Fanuc KAREL source: NC0056.KL

-- PROVISIONAL review KL for V940-1; original PC SHA256 2b6319c3cb2ebb61502ed711de4ec4e3f4f6b1a3b38024a92c039d9d4e8bd108
-- Incomplete behavior may be omitted. Consult companion uncertainty JSON. Do not deploy.
PROGRAM NC0056
%NOLOCKGROUP
-- UNRESOLVED_LOCAL_POOL 1 cells at code offset 3; source declarations unknown
-- DIRECT_LOCAL_WORD_ACCESS alone does not prove INTEGER, REAL, or BOOLEAN
BEGIN
  -- V9_CONDITION_STACK_HINT 4 bounded expression windows; static native code-base-relative target link; source arms held
  -- UNRESOLVED_PC offsets 0-8; opcodes 2B,2C,7B
  -- UNRESOLVED_PC offsets 13-20; opcodes 9D,23
  -- UNRESOLVED_PC offsets 25-42; opcodes 21,40,41,42
  -- UNRESOLVED_PC offsets 47-81; opcodes 21,2E,52,23,7A,40,41,42
  -- UNRESOLVED_PC offsets 86-110; opcodes 21,2E,52,23,7A,43
  -- UNRESOLVED_PC offsets 115-128; opcodes 21,9D,57,79
  -- UNRESOLVED_PC offsets 133-151; opcodes 21,2E,52,23
  -- UNRESOLVED_PC offsets 156-161; opcodes 7A
  -- UNRESOLVED_PC offsets 166-183; opcodes 21,40,41,42
  -- UNRESOLVED_PC offsets 188-222; opcodes 21,2E,52,23,7A,40,41,42
  -- UNRESOLVED_PC offsets 227-251; opcodes 21,2E,52,23,7A,43
  -- UNRESOLVED_PC offsets 256-269; opcodes 21,9D,57,79
  -- UNRESOLVED_PC offsets 274-292; opcodes 21,2E,52,23
  -- UNRESOLVED_PC offsets 297-302; opcodes 7A
  -- UNRESOLVED_PC offsets 307-324; opcodes 21,40,41,42
  -- UNRESOLVED_PC offsets 329-363; opcodes 21,2E,52,23,7A,40,41,42
  -- UNRESOLVED_PC offsets 368-392; opcodes 21,2E,52,23,7A,43
  -- UNRESOLVED_PC offsets 397-410; opcodes 21,9D,57,79
  -- UNRESOLVED_PC offsets 415-433; opcodes 21,2E,52,23
  -- UNRESOLVED_PC offsets 438-443; opcodes 7A
  -- UNRESOLVED_PC offsets 448-465; opcodes 21,40,41,42
  -- UNRESOLVED_PC offsets 470-504; opcodes 21,2E,52,23,7A,40,41,42
  -- UNRESOLVED_PC offsets 509-533; opcodes 21,2E,52,23,7A,43
  -- UNRESOLVED_PC offsets 538-551; opcodes 21,9D,57,79
  -- UNRESOLVED_PC offsets 556-574; opcodes 21,2E,52,23
  -- UNRESOLVED_PC offsets 579-584; opcodes 7A
  -- UNRESOLVED_PC offsets 589-603; opcodes 21,9D,52,23
  -- UNRESOLVED_PC offsets 648-652; opcodes 7F
  -- UNRESOLVED_PC offsets 657-661; opcodes 27,AA
  -- UNRESOLVED_PC offsets 666-670; opcodes 7F
END NC0056
